DECL E6POS XP595={X -550,Y 570,Z 550,A 0,B -90,C 180,S 6,T 16,E1 0.0,E2 0.0,E3 0.0,E4 0.0,E5 0.0,E6 0.0}
DECL FDAT FP595={TOOL_NO 4,BASE_NO 2,IPO_FRAME #BASE,POINT2[] " "}
DECL LDAT LCPDAT595={VEL 1,ACC 50.000,APO_DIST 500.000,APO_FAC 50.0000,AXIS_VEL 50.000,AXIS_ACC 50.000,ORI_TYP #VAR,CIRC_TYP #BASE,JERK_FAC 50.0000,GEAR_JERK 100.000,EXAX_IGN 0}

DECL E6POS XP596={X -500,Y 570,Z 550,A 0,B -90,C 180,S 6,T 16,E1 0.0,E2 0.0,E3 0.0,E4 0.0,E5 0.0,E6 0.0}
DECL FDAT FP596={TOOL_NO 4,BASE_NO 2,IPO_FRAME #BASE,POINT2[] " "}
DECL LDAT LCPDAT596={VEL 1,ACC 50.000,APO_DIST 500.000,APO_FAC 50.0000,AXIS_VEL 50.000,AXIS_ACC 50.000,ORI_TYP #VAR,CIRC_TYP #BASE,JERK_FAC 50.0000,GEAR_JERK 100.000,EXAX_IGN 0}

DECL E6POS XP597={X -450,Y 570,Z 550,A 0,B -90,C 180,S 6,T 16,E1 0.0,E2 0.0,E3 0.0,E4 0.0,E5 0.0,E6 0.0}
DECL FDAT FP597={TOOL_NO 4,BASE_NO 2,IPO_FRAME #BASE,POINT2[] " "}
DECL LDAT LCPDAT597={VEL 1,ACC 50.000,APO_DIST 500.000,APO_FAC 50.0000,AXIS_VEL 50.000,AXIS_ACC 50.000,ORI_TYP #VAR,CIRC_TYP #BASE,JERK_FAC 50.0000,GEAR_JERK 100.000,EXAX_IGN 0}

DECL E6POS XP598={X -400,Y 570,Z 550,A 0,B -90,C 180,S 6,T 16,E1 0.0,E2 0.0,E3 0.0,E4 0.0,E5 0.0,E6 0.0}
DECL FDAT FP598={TOOL_NO 4,BASE_NO 2,IPO_FRAME #BASE,POINT2[] " "}
DECL LDAT LCPDAT598={VEL 1,ACC 50.000,APO_DIST 500.000,APO_FAC 50.0000,AXIS_VEL 50.000,AXIS_ACC 50.000,ORI_TYP #VAR,CIRC_TYP #BASE,JERK_FAC 50.0000,GEAR_JERK 100.000,EXAX_IGN 0}

DECL E6POS XP599={X -350,Y 570,Z 550,A 0,B -90,C 180,S 6,T 16,E1 0.0,E2 0.0,E3 0.0,E4 0.0,E5 0.0,E6 0.0}
DECL FDAT FP599={TOOL_NO 4,BASE_NO 2,IPO_FRAME #BASE,POINT2[] " "}
DECL LDAT LCPDAT599={VEL 1,ACC 50.000,APO_DIST 500.000,APO_FAC 50.0000,AXIS_VEL 50.000,AXIS_ACC 50.000,ORI_TYP #VAR,CIRC_TYP #BASE,JERK_FAC 50.0000,GEAR_JERK 100.000,EXAX_IGN 0}

DECL E6POS XP600={X -300,Y 570,Z 550,A 0,B -90,C 180,S 6,T 16,E1 0.0,E2 0.0,E3 0.0,E4 0.0,E5 0.0,E6 0.0}
DECL FDAT FP600={TOOL_NO 4,BASE_NO 2,IPO_FRAME #BASE,POINT2[] " "}
DECL LDAT LCPDAT600={VEL 1,ACC 50.000,APO_DIST 500.000,APO_FAC 50.0000,AXIS_VEL 50.000,AXIS_ACC 50.000,ORI_TYP #VAR,CIRC_TYP #BASE,JERK_FAC 50.0000,GEAR_JERK 100.000,EXAX_IGN 0}

DECL E6POS XP601={X -250,Y 570,Z 550,A 0,B -90,C 180,S 6,T 16,E1 0.0,E2 0.0,E3 0.0,E4 0.0,E5 0.0,E6 0.0}
DECL FDAT FP601={TOOL_NO 4,BASE_NO 2,IPO_FRAME #BASE,POINT2[] " "}
DECL LDAT LCPDAT601={VEL 1,ACC 50.000,APO_DIST 500.000,APO_FAC 50.0000,AXIS_VEL 50.000,AXIS_ACC 50.000,ORI_TYP #VAR,CIRC_TYP #BASE,JERK_FAC 50.0000,GEAR_JERK 100.000,EXAX_IGN 0}

DECL E6POS XP602={X -200,Y 570,Z 550,A 0,B -90,C 180,S 6,T 16,E1 0.0,E2 0.0,E3 0.0,E4 0.0,E5 0.0,E6 0.0}
DECL FDAT FP602={TOOL_NO 4,BASE_NO 2,IPO_FRAME #BASE,POINT2[] " "}
DECL LDAT LCPDAT602={VEL 1,ACC 50.000,APO_DIST 500.000,APO_FAC 50.0000,AXIS_VEL 50.000,AXIS_ACC 50.000,ORI_TYP #VAR,CIRC_TYP #BASE,JERK_FAC 50.0000,GEAR_JERK 100.000,EXAX_IGN 0}

DECL E6POS XP603={X -150,Y 570,Z 550,A 0,B -90,C 180,S 6,T 16,E1 0.0,E2 0.0,E3 0.0,E4 0.0,E5 0.0,E6 0.0}
DECL FDAT FP603={TOOL_NO 4,BASE_NO 2,IPO_FRAME #BASE,POINT2[] " "}
DECL LDAT LCPDAT603={VEL 1,ACC 50.000,APO_DIST 500.000,APO_FAC 50.0000,AXIS_VEL 50.000,AXIS_ACC 50.000,ORI_TYP #VAR,CIRC_TYP #BASE,JERK_FAC 50.0000,GEAR_JERK 100.000,EXAX_IGN 0}

DECL E6POS XP604={X -100,Y 570,Z 550,A 0,B -90,C 180,S 6,T 16,E1 0.0,E2 0.0,E3 0.0,E4 0.0,E5 0.0,E6 0.0}
DECL FDAT FP604={TOOL_NO 4,BASE_NO 2,IPO_FRAME #BASE,POINT2[] " "}
DECL LDAT LCPDAT604={VEL 1,ACC 50.000,APO_DIST 500.000,APO_FAC 50.0000,AXIS_VEL 50.000,AXIS_ACC 50.000,ORI_TYP #VAR,CIRC_TYP #BASE,JERK_FAC 50.0000,GEAR_JERK 100.000,EXAX_IGN 0}

DECL E6POS XP605={X -50,Y 570,Z 550,A 0,B -90,C 180,S 6,T 16,E1 0.0,E2 0.0,E3 0.0,E4 0.0,E5 0.0,E6 0.0}
DECL FDAT FP605={TOOL_NO 4,BASE_NO 2,IPO_FRAME #BASE,POINT2[] " "}
DECL LDAT LCPDAT605={VEL 1,ACC 50.000,APO_DIST 500.000,APO_FAC 50.0000,AXIS_VEL 50.000,AXIS_ACC 50.000,ORI_TYP #VAR,CIRC_TYP #BASE,JERK_FAC 50.0000,GEAR_JERK 100.000,EXAX_IGN 0}

DECL E6POS XP606={X 0,Y 570,Z 550,A 0,B -90,C 180,S 6,T 16,E1 0.0,E2 0.0,E3 0.0,E4 0.0,E5 0.0,E6 0.0}
DECL FDAT FP606={TOOL_NO 4,BASE_NO 2,IPO_FRAME #BASE,POINT2[] " "}
DECL LDAT LCPDAT606={VEL 1,ACC 50.000,APO_DIST 500.000,APO_FAC 50.0000,AXIS_VEL 50.000,AXIS_ACC 50.000,ORI_TYP #VAR,CIRC_TYP #BASE,JERK_FAC 50.0000,GEAR_JERK 100.000,EXAX_IGN 0}

DECL E6POS XP607={X 0,Y 570,Z 600,A 0,B -90,C 180,S 6,T 16,E1 0.0,E2 0.0,E3 0.0,E4 0.0,E5 0.0,E6 0.0}
DECL FDAT FP607={TOOL_NO 4,BASE_NO 2,IPO_FRAME #BASE,POINT2[] " "}
DECL LDAT LCPDAT607={VEL 1,ACC 50.000,APO_DIST 500.000,APO_FAC 50.0000,AXIS_VEL 50.000,AXIS_ACC 50.000,ORI_TYP #VAR,CIRC_TYP #BASE,JERK_FAC 50.0000,GEAR_JERK 100.000,EXAX_IGN 0}

DECL E6POS XP608={X -50,Y 570,Z 600,A 0,B -90,C 180,S 6,T 16,E1 0.0,E2 0.0,E3 0.0,E4 0.0,E5 0.0,E6 0.0}
DECL FDAT FP608={TOOL_NO 4,BASE_NO 2,IPO_FRAME #BASE,POINT2[] " "}
DECL LDAT LCPDAT608={VEL 1,ACC 50.000,APO_DIST 500.000,APO_FAC 50.0000,AXIS_VEL 50.000,AXIS_ACC 50.000,ORI_TYP #VAR,CIRC_TYP #BASE,JERK_FAC 50.0000,GEAR_JERK 100.000,EXAX_IGN 0}

DECL E6POS XP609={X -100,Y 570,Z 600,A 0,B -90,C 180,S 6,T 16,E1 0.0,E2 0.0,E3 0.0,E4 0.0,E5 0.0,E6 0.0}
DECL FDAT FP609={TOOL_NO 4,BASE_NO 2,IPO_FRAME #BASE,POINT2[] " "}
DECL LDAT LCPDAT609={VEL 1,ACC 50.000,APO_DIST 500.000,APO_FAC 50.0000,AXIS_VEL 50.000,AXIS_ACC 50.000,ORI_TYP #VAR,CIRC_TYP #BASE,JERK_FAC 50.0000,GEAR_JERK 100.000,EXAX_IGN 0}

DECL E6POS XP610={X -150,Y 570,Z 600,A 0,B -90,C 180,S 6,T 16,E1 0.0,E2 0.0,E3 0.0,E4 0.0,E5 0.0,E6 0.0}
DECL FDAT FP610={TOOL_NO 4,BASE_NO 2,IPO_FRAME #BASE,POINT2[] " "}
DECL LDAT LCPDAT610={VEL 1,ACC 50.000,APO_DIST 500.000,APO_FAC 50.0000,AXIS_VEL 50.000,AXIS_ACC 50.000,ORI_TYP #VAR,CIRC_TYP #BASE,JERK_FAC 50.0000,GEAR_JERK 100.000,EXAX_IGN 0}

DECL E6POS XP611={X -200,Y 570,Z 600,A 0,B -90,C 180,S 6,T 16,E1 0.0,E2 0.0,E3 0.0,E4 0.0,E5 0.0,E6 0.0}
DECL FDAT FP611={TOOL_NO 4,BASE_NO 2,IPO_FRAME #BASE,POINT2[] " "}
DECL LDAT LCPDAT611={VEL 1,ACC 50.000,APO_DIST 500.000,APO_FAC 50.0000,AXIS_VEL 50.000,AXIS_ACC 50.000,ORI_TYP #VAR,CIRC_TYP #BASE,JERK_FAC 50.0000,GEAR_JERK 100.000,EXAX_IGN 0}

DECL E6POS XP612={X -250,Y 570,Z 600,A 0,B -90,C 180,S 6,T 16,E1 0.0,E2 0.0,E3 0.0,E4 0.0,E5 0.0,E6 0.0}
DECL FDAT FP612={TOOL_NO 4,BASE_NO 2,IPO_FRAME #BASE,POINT2[] " "}
DECL LDAT LCPDAT612={VEL 1,ACC 50.000,APO_DIST 500.000,APO_FAC 50.0000,AXIS_VEL 50.000,AXIS_ACC 50.000,ORI_TYP #VAR,CIRC_TYP #BASE,JERK_FAC 50.0000,GEAR_JERK 100.000,EXAX_IGN 0}

DECL E6POS XP613={X -300,Y 570,Z 600,A 0,B -90,C 180,S 6,T 16,E1 0.0,E2 0.0,E3 0.0,E4 0.0,E5 0.0,E6 0.0}
DECL FDAT FP613={TOOL_NO 4,BASE_NO 2,IPO_FRAME #BASE,POINT2[] " "}
DECL LDAT LCPDAT613={VEL 1,ACC 50.000,APO_DIST 500.000,APO_FAC 50.0000,AXIS_VEL 50.000,AXIS_ACC 50.000,ORI_TYP #VAR,CIRC_TYP #BASE,JERK_FAC 50.0000,GEAR_JERK 100.000,EXAX_IGN 0}

DECL E6POS XP614={X -350,Y 570,Z 600,A 0,B -90,C 180,S 6,T 16,E1 0.0,E2 0.0,E3 0.0,E4 0.0,E5 0.0,E6 0.0}
DECL FDAT FP614={TOOL_NO 4,BASE_NO 2,IPO_FRAME #BASE,POINT2[] " "}
DECL LDAT LCPDAT614={VEL 1,ACC 50.000,APO_DIST 500.000,APO_FAC 50.0000,AXIS_VEL 50.000,AXIS_ACC 50.000,ORI_TYP #VAR,CIRC_TYP #BASE,JERK_FAC 50.0000,GEAR_JERK 100.000,EXAX_IGN 0}

DECL E6POS XP615={X -400,Y 570,Z 600,A 0,B -90,C 180,S 6,T 16,E1 0.0,E2 0.0,E3 0.0,E4 0.0,E5 0.0,E6 0.0}
DECL FDAT FP615={TOOL_NO 4,BASE_NO 2,IPO_FRAME #BASE,POINT2[] " "}
DECL LDAT LCPDAT615={VEL 1,ACC 50.000,APO_DIST 500.000,APO_FAC 50.0000,AXIS_VEL 50.000,AXIS_ACC 50.000,ORI_TYP #VAR,CIRC_TYP #BASE,JERK_FAC 50.0000,GEAR_JERK 100.000,EXAX_IGN 0}

DECL E6POS XP616={X -450,Y 570,Z 600,A 0,B -90,C 180,S 6,T 16,E1 0.0,E2 0.0,E3 0.0,E4 0.0,E5 0.0,E6 0.0}
DECL FDAT FP616={TOOL_NO 4,BASE_NO 2,IPO_FRAME #BASE,POINT2[] " "}
DECL LDAT LCPDAT616={VEL 1,ACC 50.000,APO_DIST 500.000,APO_FAC 50.0000,AXIS_VEL 50.000,AXIS_ACC 50.000,ORI_TYP #VAR,CIRC_TYP #BASE,JERK_FAC 50.0000,GEAR_JERK 100.000,EXAX_IGN 0}

DECL E6POS XP617={X -500,Y 570,Z 600,A 0,B -90,C 180,S 6,T 16,E1 0.0,E2 0.0,E3 0.0,E4 0.0,E5 0.0,E6 0.0}
DECL FDAT FP617={TOOL_NO 4,BASE_NO 2,IPO_FRAME #BASE,POINT2[] " "}
DECL LDAT LCPDAT617={VEL 1,ACC 50.000,APO_DIST 500.000,APO_FAC 50.0000,AXIS_VEL 50.000,AXIS_ACC 50.000,ORI_TYP #VAR,CIRC_TYP #BASE,JERK_FAC 50.0000,GEAR_JERK 100.000,EXAX_IGN 0}

DECL E6POS XP618={X -550,Y 570,Z 600,A 0,B -90,C 180,S 6,T 16,E1 0.0,E2 0.0,E3 0.0,E4 0.0,E5 0.0,E6 0.0}
DECL FDAT FP618={TOOL_NO 4,BASE_NO 2,IPO_FRAME #BASE,POINT2[] " "}
DECL LDAT LCPDAT618={VEL 1,ACC 50.000,APO_DIST 500.000,APO_FAC 50.0000,AXIS_VEL 50.000,AXIS_ACC 50.000,ORI_TYP #VAR,CIRC_TYP #BASE,JERK_FAC 50.0000,GEAR_JERK 100.000,EXAX_IGN 0}

ENDDAT
